TYPE ST_CLEAR_ALARM EXTENDS ST_ALARM_BASE :
STRUCT
END_STRUCT
END_TYPE

(* stored: Version 1.1.0.1, ProductVersion 3.1.4026.18
   DUT ST_CLEAR_ALARM: Id {181a9ae4-dc2f-0862-07b7-3b2516518479} *)
